INTERFACE I_MotionlinxAI_Axis

PROPERTY HasFault : BOOL
GET
END_GET
END_PROPERTY

PROPERTY IsEnabled : BOOL
GET
END_GET
END_PROPERTY

PROPERTY IsReady : BOOL
GET
END_GET
END_PROPERTY

END_INTERFACE

(* stored: Version 1.1.0.1, ProductVersion 3.1.4024.16
   Itf I_MotionlinxAI_Axis: Id {c01f17c0-c2ad-4f76-b252-af9b94d50a71}
   Property HasFault: Id {52818e9e-a7e0-4abf-82aa-cd9bc2c1fc55}
   Get Get: Id {2813bc00-55c7-4383-a13d-fcfdd0e5834a}
   Property IsEnabled: Id {0a3ba106-c63b-4b0b-a679-d4fc962ef76a}
   Get Get: Id {70a929db-4764-47fd-b777-6c6f4493b29e}
   Property IsReady: Id {7a7448a9-a0d7-4964-91fc-4ebb07e41f8f}
   Get Get: Id {668cbaf3-91c8-4db7-af24-2323c7222229} *)
